// TIA Portal project "PROCESS_CONTROL_SYSTEM_PID" (V16)

(* hardware
DEVICE "S7-1200 station_1"  S7-1200 Station
   slot 0: "Rack_0"  S7-1200 Rack  Rack  V1.0
   slot 1: "PLC_1"  CPU 1214C DC/DC/DC  6ES7 214-1AG40-0XB0  V4.4
   slot 2: "AI 4x13BIT/AQ 2x14BIT_1"  6ES7 234-4HE32-0XB0  V2.1
*)

// ===== PLC "PLC_1"  CPU 1214C DC/DC/DC =====

VAR_GLOBAL   // PLC tag table "INPUTS&OUTPUTS"
   "START" AT %I0.1 : Bool;
   "PUMP" AT %Q0.0 : Bool;
   "SOLENOID_VALVE" AT %Q0.3 : Bool;
   "PRESSURE_SENSOR" AT %IW64 : Int;
   "FLOW_VALVE" AT %QW96 : Int;
   "OUTPUT_MEM" AT %MD67 : DWord;
   "SET_POINT" AT %MD20 : Real;
   "FRACTION_MEM" AT %MD24 : Real;
END_VAR

ORGANIZATION_BLOCK "Main"   // OB1, LAD, ProgramCycle
TITLE = "Main Program Sweep (Cycle)"
{ S7_Optimized_Access := 'TRUE' }
VERSION : 0.1
   VAR_INPUT
      Initial_Call : Bool;   // Initial call of this OB
      Remanence : Bool;   // =True, if remanent data are available
   END_VAR
BEGIN

REGION Network 1
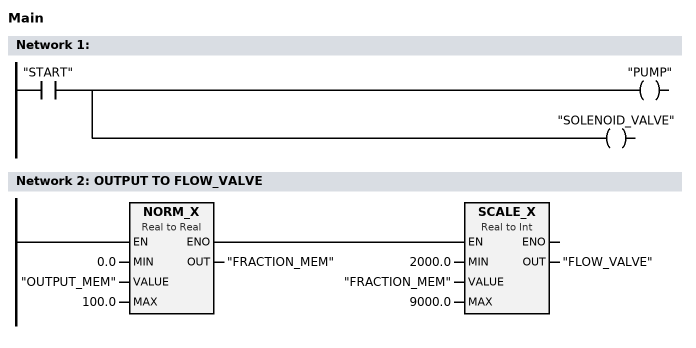
   RUNG wire#powerrail
      Contact( "START" )
      wire#w1
      Coil( "PUMP" )
   END_RUNG
   RUNG wire#w1
      Coil( "SOLENOID_VALVE" )
   END_RUNG
   // the same network as SCL:
   "PUMP" := "START";
   "SOLENOID_VALVE" := "START";
END_REGION

REGION Network 2: OUTPUT TO FLOW_VALVE
   RUNG wire#powerrail
      { S7_Templates := "[SrcType := Real, DestType := Real]" } Normalize(min := 0.0, value := "OUTPUT_MEM", max := 100.0, out => "FRACTION_MEM")
      { S7_Templates := "[SrcType := Real, DestType := Int]" } Scale(min := 2000.0, value := "FRACTION_MEM", max := 9000.0, out => "FLOW_VALVE")
   END_RUNG
   // the same network as SCL:
   "FRACTION_MEM" := NORM_X(MIN := 0.0, VALUE := "OUTPUT_MEM", MAX := 100.0);
   "FLOW_VALVE" := SCALE_X(MIN := 2000.0, VALUE := "FRACTION_MEM", MAX := 9000.0);
END_REGION
END_ORGANIZATION_BLOCK

ORGANIZATION_BLOCK "Cyclic interrupt"   // OB30, LAD, CyclicInterrupt
{ S7_Optimized_Access := 'TRUE' }
VERSION : 0.1
   VAR_INPUT
      Initial_Call : Bool;   // Initial call of this OB
      Event_Count : Int;   // Events discarded
   END_VAR
BEGIN

REGION Network 1
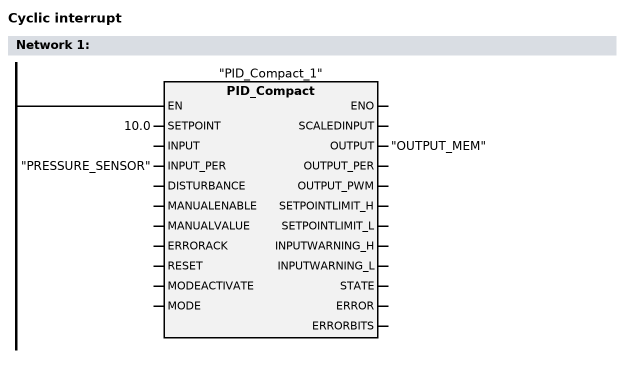
   "PID_Compact_1"(Setpoint := 10.0, Input_PER := "PRESSURE_SENSOR", Output => "OUTPUT_MEM");   // PID_Compact
END_REGION
END_ORGANIZATION_BLOCK